// TIA Portal V16 export
// export: Created 2021-08-30T10:49:32.1219073Z, ExportSetting WithDefaults, DisplayName Totally Integrated Automation Portal, DisplayVersion V16 Update 3, DisplayName TIA Portal Version Control Interface, DisplayVersion V16 Update 2, DisplayName TIA Portal Openness, DisplayVersion V16 Update 3, DisplayName TIA Portal Teamcenter Gateway, DisplayVersion V16, DisplayName STEP 7 Professional, DisplayVersion V16 Update 3, DisplayName STEP 7 Safety, DisplayVersion V16, DisplayName WinCC Advanced, DisplayVersion V16 Update 3
DATA_BLOCK "dtAV"   // DB80
{ S7_Optimized_Access := 'FALSE' }
VERSION : 0.1
// stored: AutoNumber false, DBAccessibleFromOPCUA true, IsOnlyStoredInLoadMemory false, IsWriteProtectedInAS false
   VAR RETAIN
      DVM201 { S7_SetPoint := 'True'} : "Av";
      SOV801 { S7_SetPoint := 'True'} : "Av";
      SOV901 { S7_SetPoint := 'True'} : "Av";
      SOV902 { S7_SetPoint := 'True'} : "Av";
      SOV1301 { S7_SetPoint := 'True'} : "Av";
      SOV1302 { S7_SetPoint := 'True'} : "Av";
      SOV1303 { S7_SetPoint := 'True'} : "Av";
      DVA501 { S7_SetPoint := 'True'} : "Av";
      DVA502 { S7_SetPoint := 'True'} : "Av";
      DVA504 { S7_SetPoint := 'True'} : "Av";
      DVA505 { S7_SetPoint := 'True'} : "Av";
      DVA506 { S7_SetPoint := 'True'} : "Av";
      DVA507 { S7_SetPoint := 'True'} : "Av";
      DVA508 { S7_SetPoint := 'True'} : "Av";
      DVA509 { S7_SetPoint := 'True'} : "Av";
      DVA511 { S7_SetPoint := 'True'} : "Av";
      DVA512 { S7_SetPoint := 'True'} : "Av";
      DVA513 { S7_SetPoint := 'True'} : "Av";
      DVA514 { S7_SetPoint := 'True'} : "Av";
      DVA515 { S7_SetPoint := 'True'} : "Av";
      DVA516 { S7_SetPoint := 'True'} : "Av";
      DVA1801 { S7_SetPoint := 'True'} : "Av";
   END_VAR
BEGIN
END_DATA_BLOCK
